FUNCTION_BLOCK FB_Check
VAR_INPUT
END_VAR
VAR_OUTPUT
END_VAR
VAR
	axTest: ARRAY[0..19] OF BOOL;    // Array of 20 Bool type elements
	iCell: INT;						 
	x:BOOL:=TRUE;
	iNumberOfCellWithTrueValue:INT;					// Number of cell where bool value is true
	xEndingLoop: BOOL:=FALSE;				// Variable ending loop when there is true value in array
END_VAR

// Method 
CheckIfAnyArrayElementsTrue();
// Setting values to array
IF 	NOT xEndingLoop THEN
	FOR iCell:= 0 TO 19 DO	
		// True value in 7th cell
		IF iCell = 7  THEN
			axTest[iCell]:=TRUE;
			xEndingLoop:=TRUE;
		ELSE
			axTest[iCell]:=FALSE;
		
		END_IF
	END_FOR
	xEndingLoop:=TRUE;
ELSE
	;
END_IF

METHOD CheckIfAnyArrayElementsTrue : BOOL
VAR_INPUT
END_VAR
VAR_INST
	xInArrayExistsTrueValue:BOOL;
END_VAR
// Loop ending when xCell = TRUE
IF x:=TRUE THEN
	FOR iCell:= 0 TO 19  DO
		// Searching TRUE value in array
		IF axTest[iCell]= TRUE THEN
			iNumberOfCellWithTrueValue:=iCell;
			x:=FALSE;
			xInArrayExistsTrueValue:=TRUE;
			EXIT;
		END_IF
	END_FOR
END_IF
END_METHOD

END_FUNCTION_BLOCK

(* stored: Version 1.1.0.1, ProductVersion 3.1.4024.13
   POU FB_Check: Id {d1ae89a7-59a6-47e7-974b-930426d17021}, SpecialFunc None
   Method CheckIfAnyArrayElementsTrue: Id {4438729a-5e91-4fcb-a91a-b438d3b4f5de} *)
